{attribute addProperty BoxType "EP3162-1002-0017"}
{attribute addProperty Id "Digital_outputAT %Q*ARRAY[0 ..1] OF BOOL1620"}
{attribute addProperty CRC "3842408572"}
{attribute addProperty SizeInBites "16"}
{attribute addProperty SizeInBytes "2"}
TYPE DO_Outputs_E8955222 :
STRUCT
	{attribute addProperty Name "Digital_output"}
	Digital_output AT %Q* : ARRAY[0 ..1] OF BOOL;
END_STRUCT
END_TYPE

(* stored: Version 1.2.0.0, ProductVersion 3.1.4024.9
   DUT DO_Outputs_E8955222: Id {afb9e456-a00d-4f4f-86b9-09075dad391d} *)
